TYPE U_APP_CTRL :
UNION
  stCtrl              : ST_APP_CTRL;
  byCtrl    AT %I*    : ARRAY[1..SIZEOF(ST_APP_CTRL)] OF BYTE;
END_UNION
END_TYPE

(* stored: Version 1.1.0.1, ProductVersion 3.1.4026.13
   DUT U_APP_CTRL: Id {489afe42-d50b-438f-ad3b-b903c17d0ebd} *)
